(* IEC 61131-3 sources: jiepp/tests/jiepp/input/remove_comments_option, 2 files *)

(* ---- remove_comments_option_off.iec ---- *)
/*!
 * document comment
 */

/**
 *
 */

// line comment
/* block comment 1 */
/*
block
comment
1
*/
(* block comment 2 *)
(*
block
comment
2
*)

/**
 * f
 */
function f

// line comment
/* block comment 1 */
(* block
   comment
   2 *)

end_function

//! document comment

(**
 *
 *)

(*!
 * document comment
 *)

(* ---- remove_comments_option_on.iec ---- *)
/*!
 * document comment
 */

/**
 *
 */

// line comment
/* block comment 1 */
/*
block
comment
1
*/
(* block comment 2 *)
(*
block
comment
2
*)

/**
 * f
 */
function f

// line comment
/* block comment 1 */
(* block
   comment
   2 *)

end_function

//! document comment

(**
 *
 *)

(*!
 * document comment
 *)
